FUNCTION_BLOCK FB_CylinderDiag EXTENDS FB_Cylinder
VAR_INPUT
	tTimeOut 	  : TIME;
END_VAR
VAR
	WatchDogTimer : TON;
END_VAR

;

METHOD M_Diag : BOOL
VAR_INPUT
END_VAR
IF (iState = 0) OR (iState = 3) THEN
	WatchDogTimer(IN := FALSE, PT := tTimeOut);
ELSE
	WatchDogTimer(IN := TRUE, PT := tTimeOut);
END_IF

M_Diag := WatchDogTimer.Q;
END_METHOD

METHOD M_StateMachine : BOOL
VAR_INPUT
	bPosLeftReq  : BOOL;
	bPosRightReq : BOOL;
END_VAR
VAR_OUTPUT
	bAtLeftPos  : BOOL;
	bAtRightPos : BOOL; 
END_VAR
//call M_StateMachine of base class (FB_Cylinder) via 'SUPER^.' (access to things of FB_CylinderDiag via 'THIS^.')  
SUPER^.M_StateMachine(
	bPosLeftReq 	:= bPosLeftReq,	
	bPosRightReq 	:= bPosRightReq,
	bAtLeftPos		=> bAtLeftPos,
	bAtRightPos		=> bAtRightPos,
);

//additional diagnosis
M_StateMachine 		:= M_Diag();
END_METHOD

END_FUNCTION_BLOCK

(* stored: Version 1.1.0.1, ProductVersion 3.1.4024.11
   POU FB_CylinderDiag: Id {7d5e19f8-87d2-4aed-8636-be53d03e2d7e}, SpecialFunc None
   Method M_Diag: Id {73c6a29e-1061-4f20-bdeb-4d07f65ee0d3}
   Method M_StateMachine: Id {98623343-e6a4-416f-9974-15bcd879522f} *)
